RoboDK station: clean.rdk

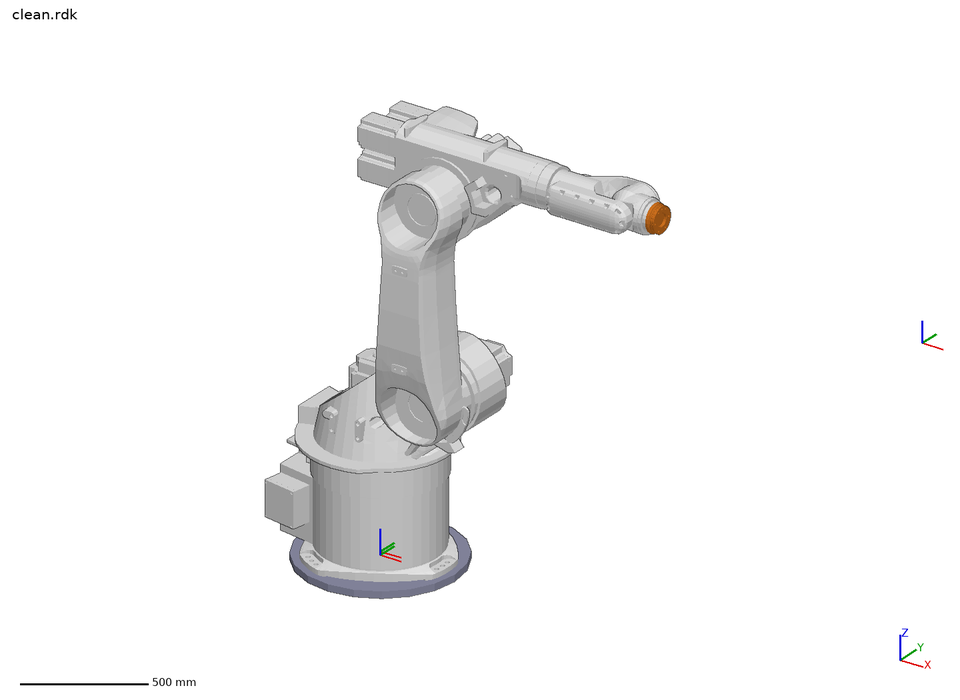
[picture v0: the station drawn from its stored meshes, robots at their saved joint values, targets as dots, program paths as lines]
Station clean. Poses are relative to the parent item; angles as X-Y-Z fixed-axis rotations.
  - frame KR 30 3 Base at (0, 0, 0) mm
    - robot KR 30 3: 6 axes
        modified DH rows (alpha deg, a mm, theta deg, d mm): 0, 0, 0, 815; -90, 350, 0, 0; 0, 850, -90, 0; -90, 145, 0, 820; 90, 0, 0, 0; -90, 0, 180, 170
        joint limits [-185, -135, -120, -350, -119, -350] to [185, 35, 158, 350, 119, 350]; home [0, -90, 90, 0, 0, 0]; saved at [0, -90, 90, 0, 0, 0]
  - frame studio at (0, 0, 0) mm
    - frame floor at (312.71, -3828.38, -30) mm
      - object x_floor at (0, 0, 0) mm, size 4780 x 9715.4 x 0 mm, geometry from x_floor.stl
    - frame post2 at (754.86, 2600, 75) mm
      - object x_post2 at (0, 0, 0) mm, size 150 x 150 x 2325 mm, geometry from x_post2.stl
    - frame post1 at (754.86, -2200, 75) mm
      - object x_post1 at (0, 0, 0) mm, size 150 x 150 x 2325 mm, geometry from x_post1.stl
    - frame girder at (670, -5360, 2630) mm
      - object x_girder at (0, 0, 0) mm, size 170.1 x 9659.7 x 304.5 mm, geometry from x_girder.stl
    - frame ceiling at (-1270, -5360, 2630) mm, rotated rx 0 ry 90 rz 0 deg
      - object x_ceiling at (0, 0, 0) mm, size 30 x 9660 x 4780 mm, geometry from x_ceiling.stl
    - frame eastWall at (-1270, -5360, 0) mm
      - object x_eastWall at (0, 0, 0) mm, size 30 x 9660 x 2630 mm, geometry from x_eastWall.stl
    - frame plinth at (0, 0, -15) mm
      - object x_plinth at (0, 0, 0) mm, size 707.6 x 707.6 x 30 mm, geometry from x_plinth.stl
  - Python program show_brush (listed below)
  - Python program draw_segment (listed below)

--- Python program show_brush ---
import sys
from robolink import (Robolink, ITEM_TYPE_ROBOT)
RL = Robolink()
brush = sys.argv[1]
robot = RL.Item('', ITEM_TYPE_ROBOT)

for c in robot.Childs():
    c.setVisible(False)

RL.Item(brush).setVisible(True)

--- Python program draw_segment ---
# Type help("robolink") or help("robodk") for more information
# Press F5 to run the script
# Documentation: https://robodk.com/doc/en/RoboDK-API.html
# Reference:     https://robodk.com/doc/en/PythonAPI/index.html
# Note: It is not required to keep a copy of this file, your python script
# is saved with the station
import sys
from robolink import (Robolink,
                      RUNMODE_SIMULATE)

import robodk as rdk    # Robot toolbox
RL = Robolink()
# sys.exit()
# mode = RL.RunMode()
# if mode != RUNMODE_SIMULATE:
#     sys.exit()

# if len(sys.argv) != 4:
#     sys.exit()

# start_mat = rdk.Mat(sys.argv[1])
# end_mat = rdk.Mat(sys.argv[2])

args = sys.argv

v0 = [float(args[1]),float(args[2]),float(args[3])]
v1 = [float(args[4]),float(args[5]),float(args[6])]
v2 = [float(args[7]),float(args[8]),float(args[9])]
v3 = [float(args[10]),float(args[11]),float(args[12])]
color = [float(args[13]),float(args[14]),float(args[15])]
name = args[16]

# verts = sys.argv[1]
# color = sys.argv[2]
# name = sys.argv[3]
# RL.ShowMessage(str(len(verts)),True)
# sys.exit()
triangles = [
    v0, v1, v2,
    v1, v3, v2
]
geo = RL.Item(name)
if not geo.Valid():
    geo = RL.AddShape(triangles)
    geo.setColor(color)
    geo.setName(name)
else:
    shape = RL.AddShape(triangles)
    shape.setColor(color)
    geo.AddGeometry(shape, rdk.eye())
    shape.Delete()
# geo.setColor(list(color))
